PROGRAM myPlcMessages
VAR
	nAirPressureValue :int;
	nCycleCounts: INT;
END_VAR

HmiMessages[0] := 'Air Pressure';
HmiMessagesValues[0] := INT_TO_STRING(nAirPressureValue);
IF nAirPressureValue < 120 THEN
	HmiMessagesColor[0] := 16#FFFF0000; // RED box
ELSE
	HmiMessagesColor[0] := 0;
END_IF

HmiMessages[1] := 'Cycle Counter';
HmiMessagesValues[1] := INT_TO_STRING(nCycleCounts);

END_PROGRAM

(* stored: Version 1.1.0.1, ProductVersion 3.1.4024.11
   POU myPlcMessages: Id {c8cfff72-9dac-49cd-bfc3-3b7d01fcc7d6}, SpecialFunc None *)
